FUNCTION_BLOCK REJ_CTL (* Peg/Ring Assembly Inspect/Reject Control *)
  (* Standard: 61499-1; Classification: Inspection; ApplicationDomain: Testbed Simulation *)
  (* Version 0.2, 2006-02-27, JHC, Holobloc Inc, Added SENSE to each transition *)
  (* Version 0.1, 2002-05-08, JHC, Rockwell Automation, Renamed inputs & outputs *)
  (* Version 0.0, 2002-04-19, JHC, Rockwell Automation *)
  (* Compiler header: package fb.rt.ita.testbed; *)
  (* Compiler Java IBM Jikes 1.06 *)
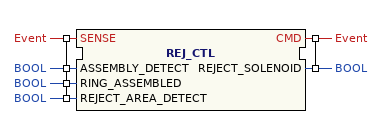
  EVENT_INPUT
    SENSE WITH ASSEMBLY_DETECT, RING_ASSEMBLED, REJECT_AREA_DETECT;
  END_EVENT
  EVENT_OUTPUT
    CMD WITH REJECT_SOLENOID;
  END_EVENT
  VAR_INPUT
    ASSEMBLY_DETECT : BOOL;
    RING_ASSEMBLED : BOOL;
    REJECT_AREA_DETECT : BOOL;
  END_VAR
  VAR_OUTPUT
    REJECT_SOLENOID : BOOL; (* REJECT SOLENOID *)
  END_VAR
  VAR
    REJ_BIT : BOOL; (* Bit to be output to REJECT_SOLENOID *)
  END_VAR
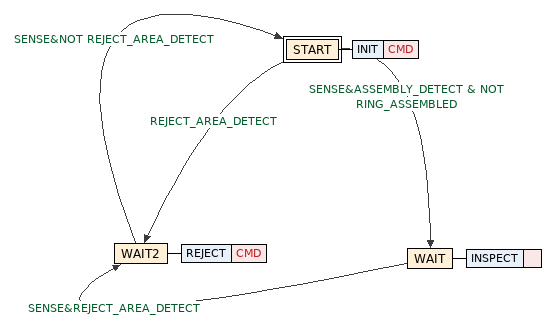
  EC_STATES
    START : INIT -> CMD; (* Waiting for Inspection *)
    WAIT : INSPECT; (* Between Inspect and Reject stations *)
    WAIT2 : REJECT -> CMD; (* Waiting to clear Reject area *)
  END_STATES
  EC_TRANSITIONS
    START TO WAIT := SENSE&ASSEMBLY_DETECT & NOT RING_ASSEMBLED;
    WAIT TO WAIT2 := SENSE&REJECT_AREA_DETECT;
    START TO WAIT2 := REJECT_AREA_DETECT;
    WAIT2 TO START := SENSE&NOT REJECT_AREA_DETECT;
  END_TRANSITIONS
  ALGORITHM INIT IN ST: (* Clear Reject Solenoid *)
REJECT_SOLENOID := FALSE;
REJ_BIT := FALSE;
  END_ALGORITHM
  ALGORITHM INSPECT IN ST: (* Inspection failed, set REJ_BIT *)
REJ_BIT := TRUE;
  END_ALGORITHM
  ALGORITHM REJECT IN ST: (* Set state of Reject Solenoid *)
REJECT_SOLENOID := REJ_BIT;
  END_ALGORITHM
END_FUNCTION_BLOCK
